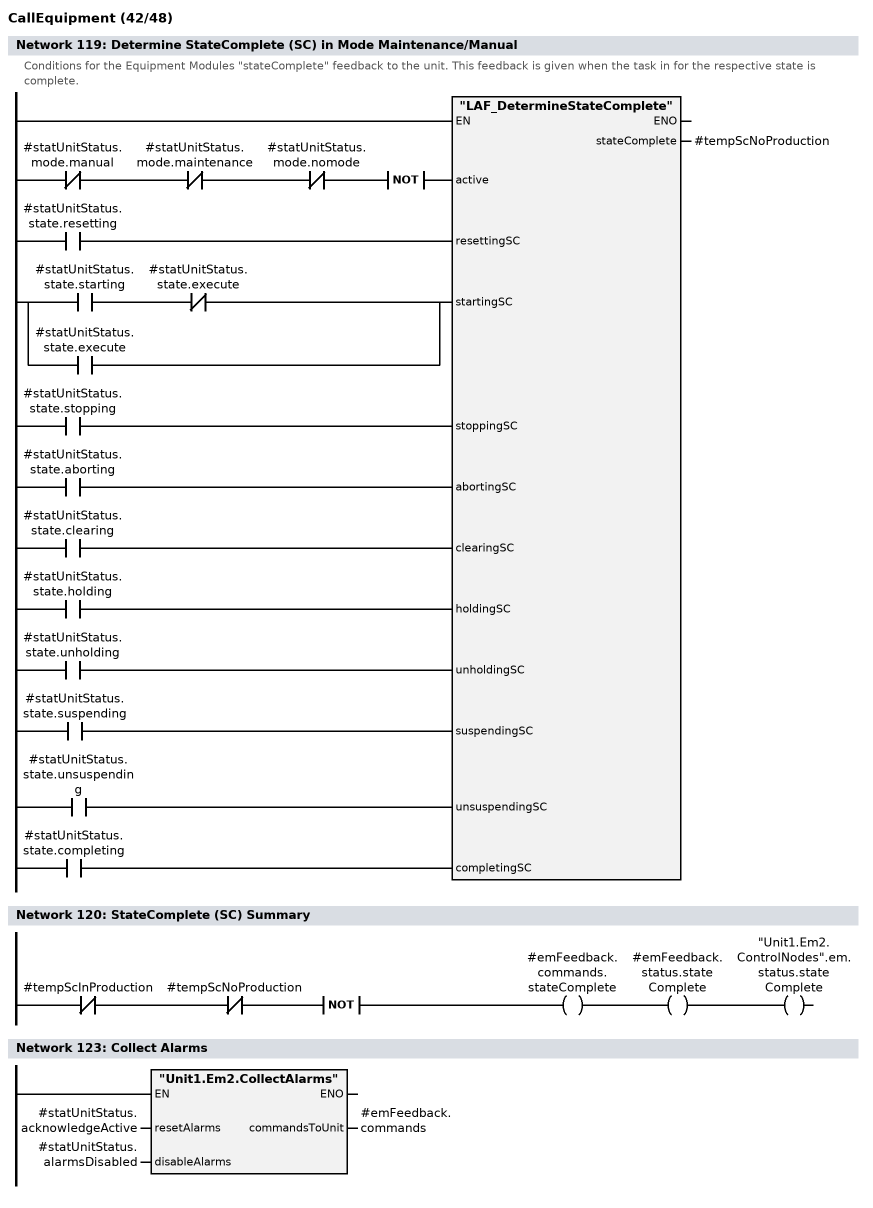
   RUNG wire#powerrail
      "LAF_DetermineStateComplete"(active := wire#w1, resettingSC := wire#w2, startingSC := wire#w3, stoppingSC := wire#w4, abortingSC := wire#w5, clearingSC := wire#w6, holdingSC := wire#w7, unholdingSC := wire#w8, suspendingSC := wire#w9, unsuspendingSC := wire#w10, completingSC := wire#w11, stateComplete => #tempScNoProduction)
   END_RUNG
   RUNG wire#powerrail
      I_Contact( #statUnitStatus.mode.manual )
      I_Contact( #statUnitStatus.mode.maintenance )
      I_Contact( #statUnitStatus.mode.nomode )
      Not()
   END_RUNG wire#w1
   RUNG wire#powerrail
      Contact( #statUnitStatus.state.resetting )
   END_RUNG wire#w2
   RUNG wire#powerrail
      Contact( #statUnitStatus.state.starting )
      I_Contact( #statUnitStatus.state.execute )
   END_RUNG wire#w3
   RUNG wire#powerrail
      Contact( #statUnitStatus.state.execute )
   END_RUNG wire#w3
   RUNG wire#powerrail
      Contact( #statUnitStatus.state.stopping )
   END_RUNG wire#w4
   RUNG wire#powerrail
      Contact( #statUnitStatus.state.aborting )
   END_RUNG wire#w5
   RUNG wire#powerrail
      Contact( #statUnitStatus.state.clearing )
   END_RUNG wire#w6
   RUNG wire#powerrail
      Contact( #statUnitStatus.state.holding )
   END_RUNG wire#w7
   RUNG wire#powerrail
      Contact( #statUnitStatus.state.unholding )
   END_RUNG wire#w8
   RUNG wire#powerrail
      Contact( #statUnitStatus.state.suspending )
   END_RUNG wire#w9
   RUNG wire#powerrail
      Contact( #statUnitStatus.state.unsuspending )
   END_RUNG wire#w10
   RUNG wire#powerrail
      Contact( #statUnitStatus.state.completing )
   END_RUNG wire#w11
   // the same network as SCL:
   "LAF_DetermineStateComplete"(active := NOT (NOT #statUnitStatus.mode.manual AND NOT #statUnitStatus.mode.maintenance AND NOT #statUnitStatus.mode.nomode),
                           resettingSC := #statUnitStatus.state.resetting,
                           startingSC := (#statUnitStatus.state.starting AND NOT #statUnitStatus.state.execute) OR #statUnitStatus.state.execute,
                           stoppingSC := #statUnitStatus.state.stopping,
                           abortingSC := #statUnitStatus.state.aborting,
                           clearingSC := #statUnitStatus.state.clearing,
                           holdingSC := #statUnitStatus.state.holding,
                           unholdingSC := #statUnitStatus.state.unholding,
                           suspendingSC := #statUnitStatus.state.suspending,
                           unsuspendingSC := #statUnitStatus.state.unsuspending,
                           completingSC := #statUnitStatus.state.completing,
                           stateComplete => #tempScNoProduction);
END_REGION

REGION Network 120: StateComplete (SC) Summary
   RUNG wire#powerrail
      I_Contact( #tempScInProduction )
      I_Contact( #tempScNoProduction )
      Not()
      Coil( #emFeedback.commands.stateComplete )
      Coil( #emFeedback.status.stateComplete )
      Coil( "Unit1.Em2.ControlNodes".em.status.stateComplete )
   END_RUNG
   // the same network as SCL:
   #emFeedback.commands.stateComplete := NOT (NOT #tempScInProduction AND NOT #tempScNoProduction);
   #emFeedback.status.stateComplete := #emFeedback.commands.stateComplete;
   "Unit1.Em2.ControlNodes".em.status.stateComplete := #emFeedback.commands.stateComplete;
END_REGION

REGION Network 122: *************** Alarms **********************************
END_REGION

REGION Network 123: Collect Alarms
   RUNG wire#powerrail
      "Unit1.Em2.CollectAlarms"(resetAlarms := #statUnitStatus.acknowledgeActive, disableAlarms := #statUnitStatus.alarmsDisabled, commandsToUnit => #emFeedback.commands)
   END_RUNG
   // the same network as SCL:
   "Unit1.Em2.CollectAlarms"(resetAlarms := #statUnitStatus.acknowledgeActive,
                           disableAlarms := #statUnitStatus.alarmsDisabled,
                           commandsToUnit => #emFeedback.commands);
END_REGION

REGION Network 124: Manage Alarms
   // Derive commands from the ProDiag supervision. The ProDiag supervisions contain categories which define the reaction of these supervisions (e.g. abort, stop, hold). These are handed over as commands to the unit level.
   // Alternatively, if no ProDiag should be used, you can use the LAF_ManageBitAlarms to realize bit alarm handling. This block can be found in LAF in folder 70_AlarmHandling.
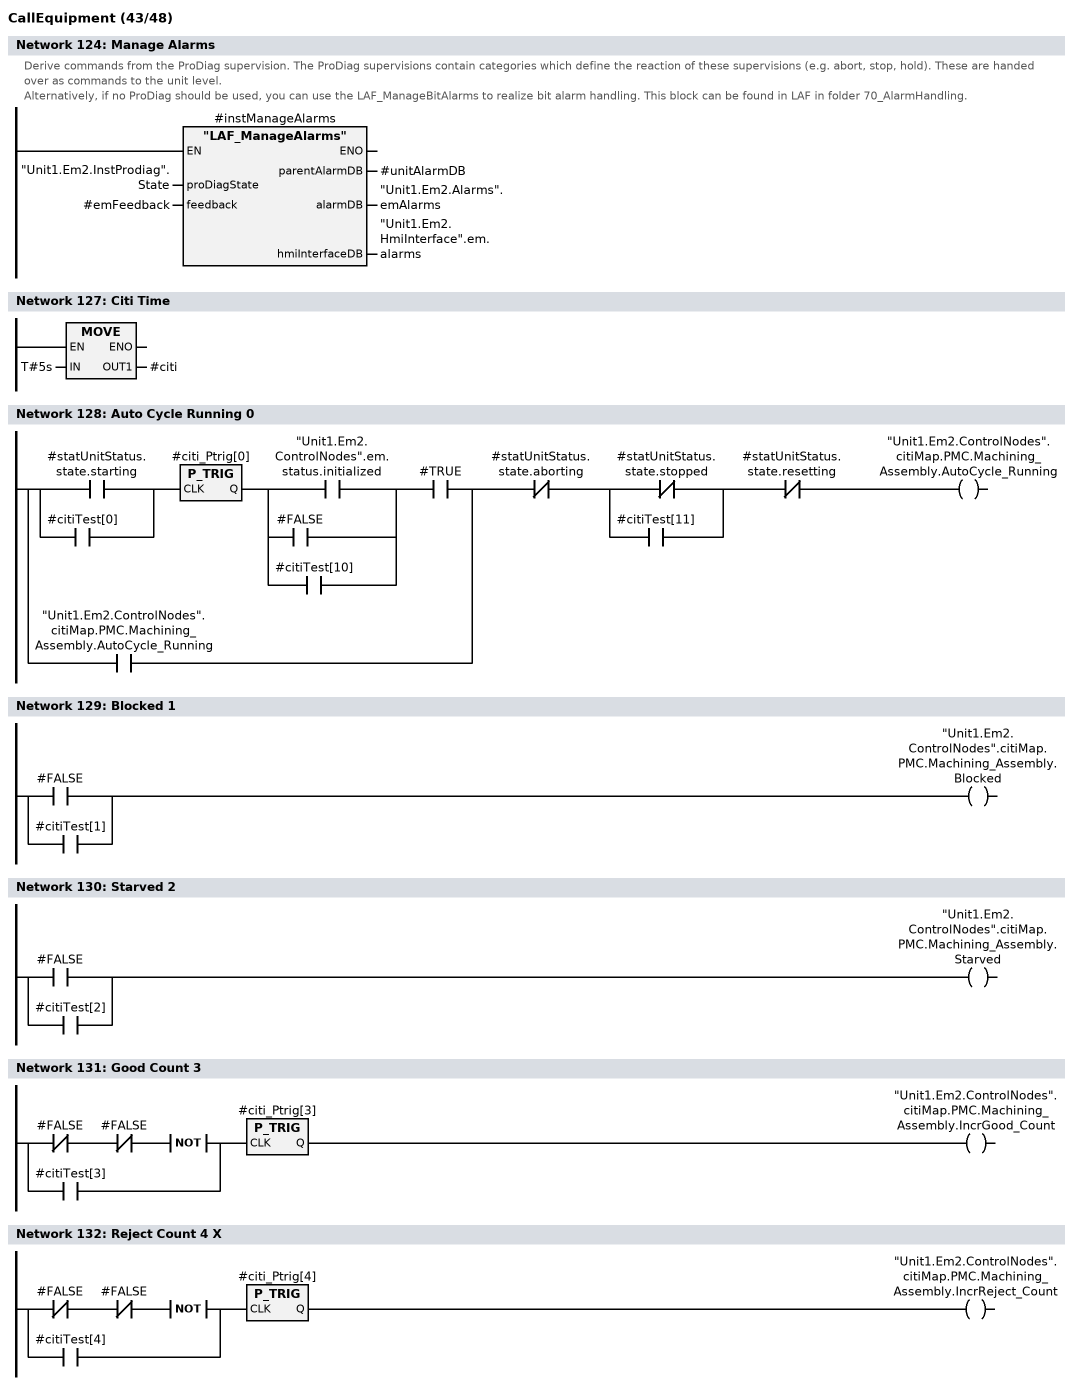
   RUNG wire#powerrail
      #instManageAlarms(proDiagState := "Unit1.Em2.InstProdiag".State, feedback := #emFeedback, parentAlarmDB => #unitAlarmDB, alarmDB => "Unit1.Em2.Alarms".emAlarms, hmiInterfaceDB => "Unit1.Em2.HmiInterface".em.alarms)
   END_RUNG
   // the same network as SCL:
   #instManageAlarms(proDiagState := "Unit1.Em2.InstProdiag".State,   // "LAF_ManageAlarms"
                     feedback := #emFeedback,
                     parentAlarmDB => #unitAlarmDB,
                     alarmDB => "Unit1.Em2.Alarms".emAlarms,
                     hmiInterfaceDB => "Unit1.Em2.HmiInterface".em.alarms);
END_REGION

REGION Network 126: ******************** CITI ********************
END_REGION

REGION Network 127: Citi Time
   RUNG wire#powerrail
      Move(in := T#5s, out1 => #citi)
   END_RUNG
   // the same network as SCL:
   #citi := T#5s;
END_REGION

REGION Network 128: Auto Cycle Running 0
   RUNG wire#powerrail
      Contact( #statUnitStatus.state.starting )
      wire#w1
      P_Trig( #citi_Ptrig[0] )
      wire#w2
      Contact( "Unit1.Em2.ControlNodes".em.status.initialized )
      wire#w3
      Contact( #TRUE )
      wire#w4
      I_Contact( #statUnitStatus.state.aborting )
      wire#w5
      I_Contact( #statUnitStatus.state.stopped )
      wire#w6
      I_Contact( #statUnitStatus.state.resetting )
      Coil( "Unit1.Em2.ControlNodes".citiMap.PMC.Machining_Assembly.AutoCycle_Running )
   END_RUNG
   RUNG wire#powerrail
      Contact( #citiTest[0] )
   END_RUNG wire#w1
   RUNG wire#w2
      Contact( #FALSE )
   END_RUNG wire#w3
   RUNG wire#w2
      Contact( #citiTest[10] )
   END_RUNG wire#w3
   RUNG wire#powerrail
      Contact( "Unit1.Em2.ControlNodes".citiMap.PMC.Machining_Assembly.AutoCycle_Running )
   END_RUNG wire#w4
   RUNG wire#w5
      Contact( #citiTest[11] )
   END_RUNG wire#w6
   // the same network as SCL:
   #_w1 := #statUnitStatus.state.starting OR #citiTest[0];
   #_w2 := #_w1 AND NOT #citi_Ptrig[0];   // rising edge
   #citi_Ptrig[0] := #_w1;
   "Unit1.Em2.ControlNodes".citiMap.PMC.Machining_Assembly.AutoCycle_Running := ((#_w2 AND ("Unit1.Em2.ControlNodes".em.status.initialized OR #FALSE OR #citiTest[10]) AND #TRUE) OR "Unit1.Em2.ControlNodes".citiMap.PMC.Machining_Assembly.AutoCycle_Running) AND NOT #statUnitStatus.state.aborting AND (NOT #statUnitStatus.state.stopped OR #citiTest[11]) AND NOT #statUnitStatus.state.resetting;
END_REGION

REGION Network 129: Blocked 1
   RUNG wire#powerrail
      Contact( #FALSE )
      wire#w1
      Coil( "Unit1.Em2.ControlNodes".citiMap.PMC.Machining_Assembly.Blocked )
   END_RUNG
   RUNG wire#powerrail
      Contact( #citiTest[1] )
   END_RUNG wire#w1
   // the same network as SCL:
   "Unit1.Em2.ControlNodes".citiMap.PMC.Machining_Assembly.Blocked := #FALSE OR #citiTest[1];
END_REGION

REGION Network 130: Starved 2
   RUNG wire#powerrail
      Contact( #FALSE )
      wire#w1
      Coil( "Unit1.Em2.ControlNodes".citiMap.PMC.Machining_Assembly.Starved )
   END_RUNG
   RUNG wire#powerrail
      Contact( #citiTest[2] )
   END_RUNG wire#w1
   // the same network as SCL:
   "Unit1.Em2.ControlNodes".citiMap.PMC.Machining_Assembly.Starved := #FALSE OR #citiTest[2];
END_REGION

REGION Network 131: Good Count 3
   RUNG wire#powerrail
      I_Contact( #FALSE )
      I_Contact( #FALSE )
      Not()
      wire#w1
      P_Trig( #citi_Ptrig[3] )
      Coil( "Unit1.Em2.ControlNodes".citiMap.PMC.Machining_Assembly.IncrGood_Count )
   END_RUNG
   RUNG wire#powerrail
      Contact( #citiTest[3] )
   END_RUNG wire#w1
   // the same network as SCL:
   #_w1 := NOT (NOT #FALSE AND NOT #FALSE) OR #citiTest[3];
   #_w2 := #_w1 AND NOT #citi_Ptrig[3];   // rising edge
   #citi_Ptrig[3] := #_w1;
   "Unit1.Em2.ControlNodes".citiMap.PMC.Machining_Assembly.IncrGood_Count := #_w2;
END_REGION

REGION Network 132: Reject Count 4 X
   RUNG wire#powerrail
      I_Contact( #FALSE )
      I_Contact( #FALSE )
      Not()
      wire#w1
      P_Trig( #citi_Ptrig[4] )
      Coil( "Unit1.Em2.ControlNodes".citiMap.PMC.Machining_Assembly.IncrReject_Count )
   END_RUNG
   RUNG wire#powerrail
      Contact( #citiTest[4] )
   END_RUNG wire#w1
   // the same network as SCL:
   #_w1 := NOT (NOT #FALSE AND NOT #FALSE) OR #citiTest[4];
   #_w2 := #_w1 AND NOT #citi_Ptrig[4];   // rising edge
   #citi_Ptrig[4] := #_w1;
   "Unit1.Em2.ControlNodes".citiMap.PMC.Machining_Assembly.IncrReject_Count := #_w2;
END_REGION

REGION Network 133: Cycle End Trigger 5
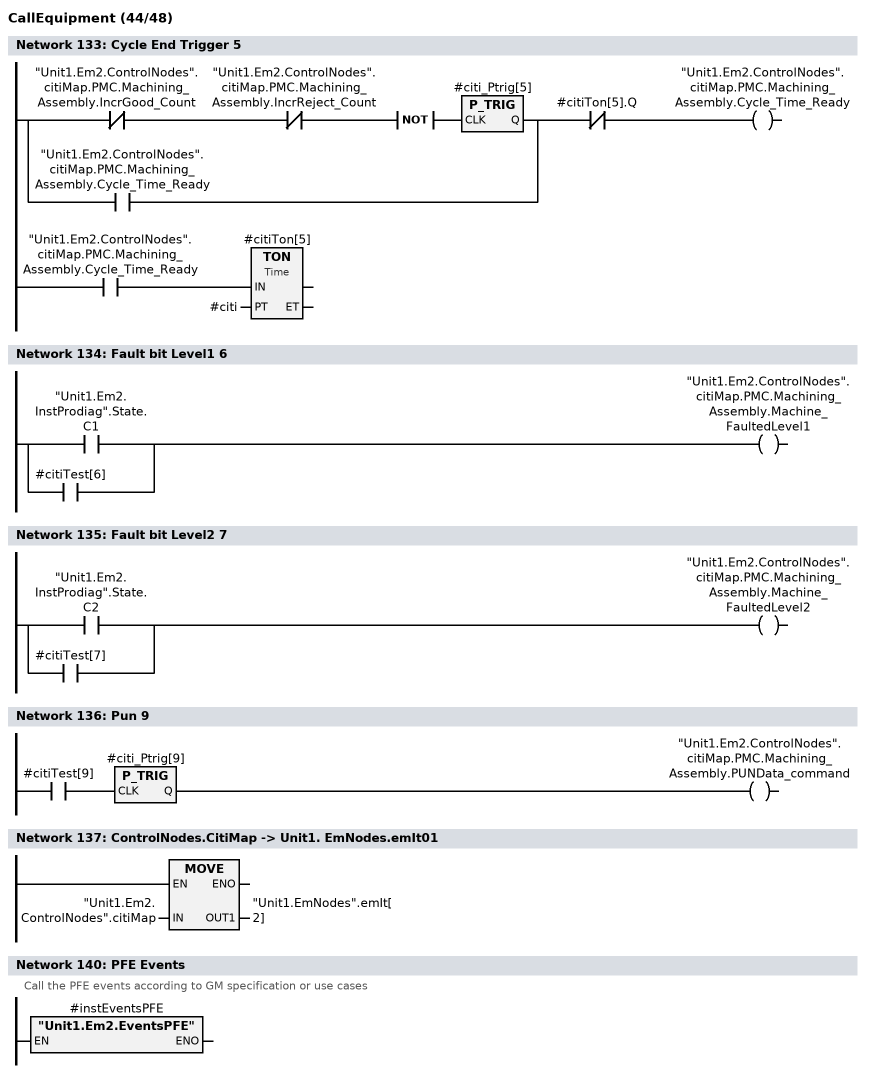
   RUNG wire#powerrail
      I_Contact( "Unit1.Em2.ControlNodes".citiMap.PMC.Machining_Assembly.IncrGood_Count )
      I_Contact( "Unit1.Em2.ControlNodes".citiMap.PMC.Machining_Assembly.IncrReject_Count )
      Not()
      P_Trig( #citi_Ptrig[5] )
      wire#w1
      I_Contact( #citiTon[5].Q )
      Coil( "Unit1.Em2.ControlNodes".citiMap.PMC.Machining_Assembly.Cycle_Time_Ready )
   END_RUNG
   RUNG wire#powerrail
      Contact( "Unit1.Em2.ControlNodes".citiMap.PMC.Machining_Assembly.Cycle_Time_Ready )
   END_RUNG wire#w1
   RUNG wire#powerrail
      Contact( "Unit1.Em2.ControlNodes".citiMap.PMC.Machining_Assembly.Cycle_Time_Ready )
      { S7_Templates := "time_type := Time" } #citiTon[5].TON(pt := #citi, et =>)
   END_RUNG
   // the same network as SCL:
   #_w1 := NOT (NOT "Unit1.Em2.ControlNodes".citiMap.PMC.Machining_Assembly.IncrGood_Count AND NOT "Unit1.Em2.ControlNodes".citiMap.PMC.Machining_Assembly.IncrReject_Count);
   #_w2 := #_w1 AND NOT #citi_Ptrig[5];   // rising edge
   #citi_Ptrig[5] := #_w1;
   "Unit1.Em2.ControlNodes".citiMap.PMC.Machining_Assembly.Cycle_Time_Ready := (#_w2 OR "Unit1.Em2.ControlNodes".citiMap.PMC.Machining_Assembly.Cycle_Time_Ready) AND NOT #citiTon[5].Q;
   #citiTon[5].TON(IN := "Unit1.Em2.ControlNodes".citiMap.PMC.Machining_Assembly.Cycle_Time_Ready, PT := #citi);
END_REGION

REGION Network 134: Fault bit Level1 6
   RUNG wire#powerrail
      Contact( "Unit1.Em2.InstProdiag".State.C1 )
      wire#w1
      Coil( "Unit1.Em2.ControlNodes".citiMap.PMC.Machining_Assembly.Machine_FaultedLevel1 )
   END_RUNG
   RUNG wire#powerrail
      Contact( #citiTest[6] )
   END_RUNG wire#w1
   // the same network as SCL:
   "Unit1.Em2.ControlNodes".citiMap.PMC.Machining_Assembly.Machine_FaultedLevel1 := "Unit1.Em2.InstProdiag".State.C1 OR #citiTest[6];
END_REGION

REGION Network 135: Fault bit Level2 7
   RUNG wire#powerrail
      Contact( "Unit1.Em2.InstProdiag".State.C2 )
      wire#w1
      Coil( "Unit1.Em2.ControlNodes".citiMap.PMC.Machining_Assembly.Machine_FaultedLevel2 )
   END_RUNG
   RUNG wire#powerrail
      Contact( #citiTest[7] )
   END_RUNG wire#w1
   // the same network as SCL:
   "Unit1.Em2.ControlNodes".citiMap.PMC.Machining_Assembly.Machine_FaultedLevel2 := "Unit1.Em2.InstProdiag".State.C2 OR #citiTest[7];
END_REGION

REGION Network 136: Pun 9
   RUNG wire#powerrail
      Contact( #citiTest[9] )
      P_Trig( #citi_Ptrig[9] )
      Coil( "Unit1.Em2.ControlNodes".citiMap.PMC.Machining_Assembly.PUNData_command )
   END_RUNG
   // the same network as SCL:
   #_w1 := #citiTest[9] AND NOT #citi_Ptrig[9];   // rising edge
   #citi_Ptrig[9] := #citiTest[9];
   "Unit1.Em2.ControlNodes".citiMap.PMC.Machining_Assembly.PUNData_command := #_w1;
END_REGION

REGION Network 137: ControlNodes.CitiMap -> Unit1. EmNodes.emIt01
   RUNG wire#powerrail
      Move(in := "Unit1.Em2.ControlNodes".citiMap, out1 => "Unit1.EmNodes".emIt[2])
   END_RUNG
   // the same network as SCL:
   "Unit1.EmNodes".emIt[2] := "Unit1.Em2.ControlNodes".citiMap;
END_REGION

REGION Network 139: *************** PFE Events**********************************
END_REGION

REGION Network 140: PFE Events
   // Call the PFE events according to GM specification or use cases
   RUNG wire#powerrail
      #instEventsPFE()
   END_RUNG
   // the same network as SCL:
   #instEventsPFE();   // "Unit1.Em2.EventsPFE"
END_REGION

REGION Network 142: ******************** Unit Output ********************
END_REGION

REGION Network 143: Em2 Relations Softcam
END_REGION

REGION Network 144: Em2 Relations Home Check
END_REGION

REGION Network 145: Em2 Relations Cm Status Cylinder
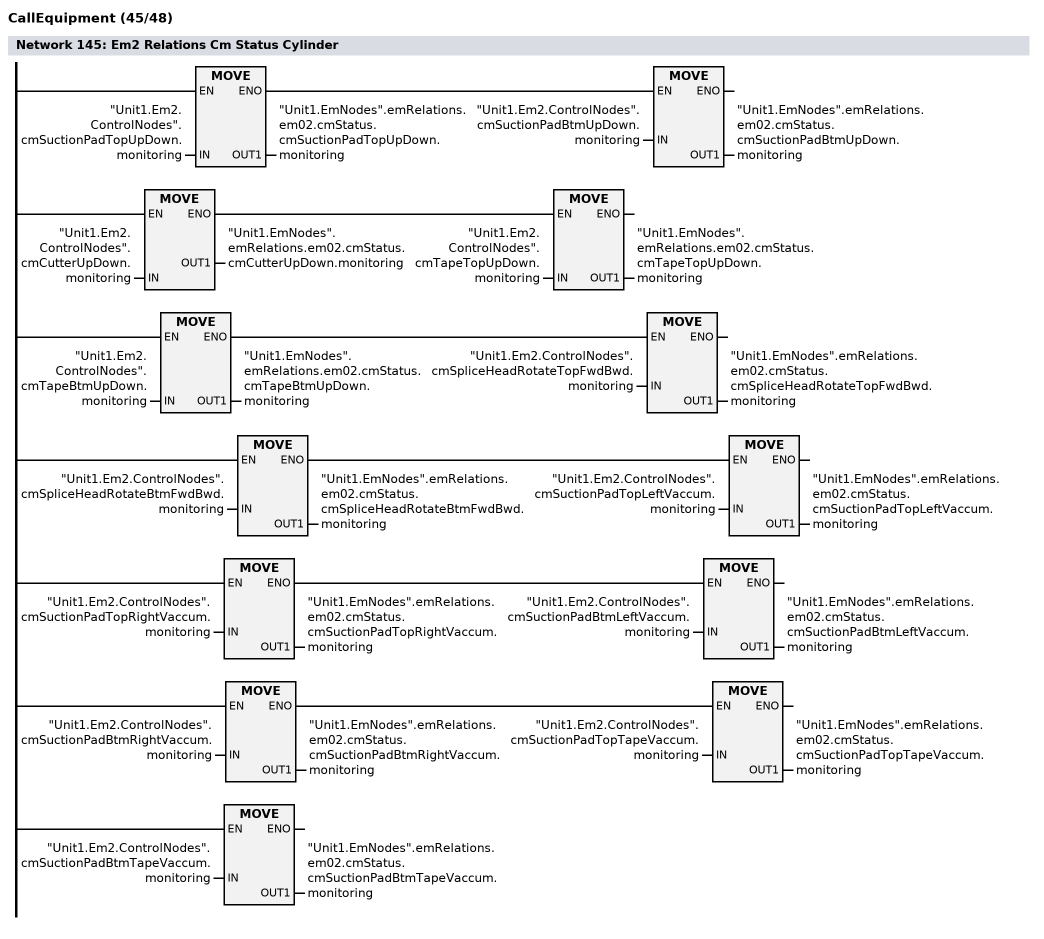
   RUNG wire#powerrail
      Move(in := "Unit1.Em2.ControlNodes".cmSuctionPadTopUpDown.monitoring, out1 => "Unit1.EmNodes".emRelations.em02.cmStatus.cmSuctionPadTopUpDown.monitoring)
      Move(in := "Unit1.Em2.ControlNodes".cmSuctionPadBtmUpDown.monitoring, out1 => "Unit1.EmNodes".emRelations.em02.cmStatus.cmSuctionPadBtmUpDown.monitoring)
   END_RUNG
   RUNG wire#powerrail
      Move(in := "Unit1.Em2.ControlNodes".cmCutterUpDown.monitoring, out1 => "Unit1.EmNodes".emRelations.em02.cmStatus.cmCutterUpDown.monitoring)
      Move(in := "Unit1.Em2.ControlNodes".cmTapeTopUpDown.monitoring, out1 => "Unit1.EmNodes".emRelations.em02.cmStatus.cmTapeTopUpDown.monitoring)
   END_RUNG
   RUNG wire#powerrail
      Move(in := "Unit1.Em2.ControlNodes".cmTapeBtmUpDown.monitoring, out1 => "Unit1.EmNodes".emRelations.em02.cmStatus.cmTapeBtmUpDown.monitoring)
      Move(in := "Unit1.Em2.ControlNodes".cmSpliceHeadRotateTopFwdBwd.monitoring, out1 => "Unit1.EmNodes".emRelations.em02.cmStatus.cmSpliceHeadRotateTopFwdBwd.monitoring)
   END_RUNG
   RUNG wire#powerrail
      Move(in := "Unit1.Em2.ControlNodes".cmSpliceHeadRotateBtmFwdBwd.monitoring, out1 => "Unit1.EmNodes".emRelations.em02.cmStatus.cmSpliceHeadRotateBtmFwdBwd.monitoring)
      Move(in := "Unit1.Em2.ControlNodes".cmSuctionPadTopLeftVaccum.monitoring, out1 => "Unit1.EmNodes".emRelations.em02.cmStatus.cmSuctionPadTopLeftVaccum.monitoring)
   END_RUNG
   RUNG wire#powerrail
      Move(in := "Unit1.Em2.ControlNodes".cmSuctionPadTopRightVaccum.monitoring, out1 => "Unit1.EmNodes".emRelations.em02.cmStatus.cmSuctionPadTopRightVaccum.monitoring)
      Move(in := "Unit1.Em2.ControlNodes".cmSuctionPadBtmLeftVaccum.monitoring, out1 => "Unit1.EmNodes".emRelations.em02.cmStatus.cmSuctionPadBtmLeftVaccum.monitoring)
   END_RUNG
   RUNG wire#powerrail
      Move(in := "Unit1.Em2.ControlNodes".cmSuctionPadBtmRightVaccum.monitoring, out1 => "Unit1.EmNodes".emRelations.em02.cmStatus.cmSuctionPadBtmRightVaccum.monitoring)
      Move(in := "Unit1.Em2.ControlNodes".cmSuctionPadTopTapeVaccum.monitoring, out1 => "Unit1.EmNodes".emRelations.em02.cmStatus.cmSuctionPadTopTapeVaccum.monitoring)
   END_RUNG
   RUNG wire#powerrail
      Move(in := "Unit1.Em2.ControlNodes".cmSuctionPadBtmTapeVaccum.monitoring, out1 => "Unit1.EmNodes".emRelations.em02.cmStatus.cmSuctionPadBtmTapeVaccum.monitoring)
   END_RUNG
   // the same network as SCL:
   "Unit1.EmNodes".emRelations.em02.cmStatus.cmSuctionPadTopUpDown.monitoring := "Unit1.Em2.ControlNodes".cmSuctionPadTopUpDown.monitoring;
   "Unit1.EmNodes".emRelations.em02.cmStatus.cmSuctionPadBtmUpDown.monitoring := "Unit1.Em2.ControlNodes".cmSuctionPadBtmUpDown.monitoring;
   "Unit1.EmNodes".emRelations.em02.cmStatus.cmCutterUpDown.monitoring := "Unit1.Em2.ControlNodes".cmCutterUpDown.monitoring;
   "Unit1.EmNodes".emRelations.em02.cmStatus.cmTapeTopUpDown.monitoring := "Unit1.Em2.ControlNodes".cmTapeTopUpDown.monitoring;
   "Unit1.EmNodes".emRelations.em02.cmStatus.cmTapeBtmUpDown.monitoring := "Unit1.Em2.ControlNodes".cmTapeBtmUpDown.monitoring;
   "Unit1.EmNodes".emRelations.em02.cmStatus.cmSpliceHeadRotateTopFwdBwd.monitoring := "Unit1.Em2.ControlNodes".cmSpliceHeadRotateTopFwdBwd.monitoring;
   "Unit1.EmNodes".emRelations.em02.cmStatus.cmSpliceHeadRotateBtmFwdBwd.monitoring := "Unit1.Em2.ControlNodes".cmSpliceHeadRotateBtmFwdBwd.monitoring;
   "Unit1.EmNodes".emRelations.em02.cmStatus.cmSuctionPadTopLeftVaccum.monitoring := "Unit1.Em2.ControlNodes".cmSuctionPadTopLeftVaccum.monitoring;
   "Unit1.EmNodes".emRelations.em02.cmStatus.cmSuctionPadTopRightVaccum.monitoring := "Unit1.Em2.ControlNodes".cmSuctionPadTopRightVaccum.monitoring;
   "Unit1.EmNodes".emRelations.em02.cmStatus.cmSuctionPadBtmLeftVaccum.monitoring := "Unit1.Em2.ControlNodes".cmSuctionPadBtmLeftVaccum.monitoring;
   "Unit1.EmNodes".emRelations.em02.cmStatus.cmSuctionPadBtmRightVaccum.monitoring := "Unit1.Em2.ControlNodes".cmSuctionPadBtmRightVaccum.monitoring;
   "Unit1.EmNodes".emRelations.em02.cmStatus.cmSuctionPadTopTapeVaccum.monitoring := "Unit1.Em2.ControlNodes".cmSuctionPadTopTapeVaccum.monitoring;
   "Unit1.EmNodes".emRelations.em02.cmStatus.cmSuctionPadBtmTapeVaccum.monitoring := "Unit1.Em2.ControlNodes".cmSuctionPadBtmTapeVaccum.monitoring;
END_REGION

REGION Network 146: Em2 Relations CmStatus Digital Signal
END_REGION

REGION Network 147: Em2 Relations Select Job Status
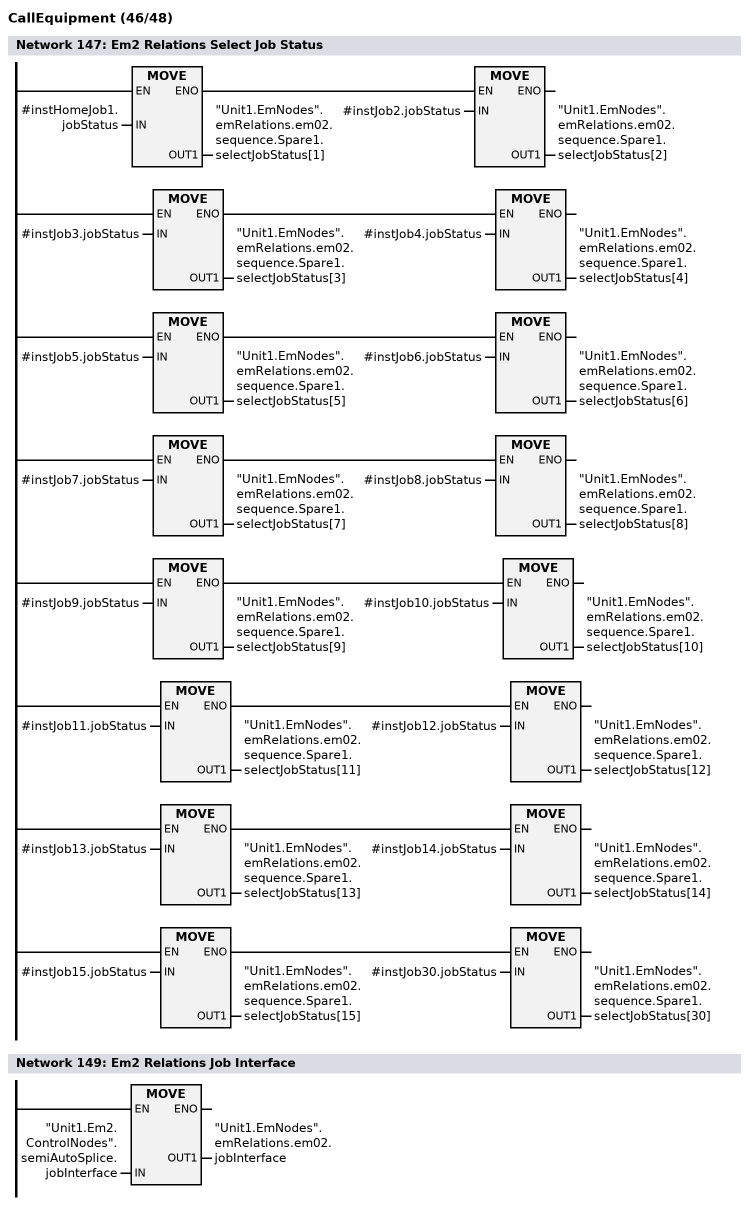
   RUNG wire#powerrail
      Move(in := #instHomeJob1.jobStatus, out1 => "Unit1.EmNodes".emRelations.em02.sequence.Spare1.selectJobStatus[1])
      Move(in := #instJob2.jobStatus, out1 => "Unit1.EmNodes".emRelations.em02.sequence.Spare1.selectJobStatus[2])
   END_RUNG
   RUNG wire#powerrail
      Move(in := #instJob3.jobStatus, out1 => "Unit1.EmNodes".emRelations.em02.sequence.Spare1.selectJobStatus[3])
      Move(in := #instJob4.jobStatus, out1 => "Unit1.EmNodes".emRelations.em02.sequence.Spare1.selectJobStatus[4])
   END_RUNG
   RUNG wire#powerrail
      Move(in := #instJob5.jobStatus, out1 => "Unit1.EmNodes".emRelations.em02.sequence.Spare1.selectJobStatus[5])
      Move(in := #instJob6.jobStatus, out1 => "Unit1.EmNodes".emRelations.em02.sequence.Spare1.selectJobStatus[6])
   END_RUNG
   RUNG wire#powerrail
      Move(in := #instJob7.jobStatus, out1 => "Unit1.EmNodes".emRelations.em02.sequence.Spare1.selectJobStatus[7])
      Move(in := #instJob8.jobStatus, out1 => "Unit1.EmNodes".emRelations.em02.sequence.Spare1.selectJobStatus[8])
   END_RUNG
   RUNG wire#powerrail
      Move(in := #instJob9.jobStatus, out1 => "Unit1.EmNodes".emRelations.em02.sequence.Spare1.selectJobStatus[9])
      Move(in := #instJob10.jobStatus, out1 => "Unit1.EmNodes".emRelations.em02.sequence.Spare1.selectJobStatus[10])
   END_RUNG
   RUNG wire#powerrail
      Move(in := #instJob11.jobStatus, out1 => "Unit1.EmNodes".emRelations.em02.sequence.Spare1.selectJobStatus[11])
      Move(in := #instJob12.jobStatus, out1 => "Unit1.EmNodes".emRelations.em02.sequence.Spare1.selectJobStatus[12])
   END_RUNG
   RUNG wire#powerrail
      Move(in := #instJob13.jobStatus, out1 => "Unit1.EmNodes".emRelations.em02.sequence.Spare1.selectJobStatus[13])
      Move(in := #instJob14.jobStatus, out1 => "Unit1.EmNodes".emRelations.em02.sequence.Spare1.selectJobStatus[14])
   END_RUNG
   RUNG wire#powerrail
      Move(in := #instJob15.jobStatus, out1 => "Unit1.EmNodes".emRelations.em02.sequence.Spare1.selectJobStatus[15])
      Move(in := #instJob30.jobStatus, out1 => "Unit1.EmNodes".emRelations.em02.sequence.Spare1.selectJobStatus[30])
   END_RUNG
   // the same network as SCL:
   "Unit1.EmNodes".emRelations.em02.sequence.Spare1.selectJobStatus[1] := #instHomeJob1.jobStatus;
   "Unit1.EmNodes".emRelations.em02.sequence.Spare1.selectJobStatus[2] := #instJob2.jobStatus;
   "Unit1.EmNodes".emRelations.em02.sequence.Spare1.selectJobStatus[3] := #instJob3.jobStatus;
   "Unit1.EmNodes".emRelations.em02.sequence.Spare1.selectJobStatus[4] := #instJob4.jobStatus;
   "Unit1.EmNodes".emRelations.em02.sequence.Spare1.selectJobStatus[5] := #instJob5.jobStatus;
   "Unit1.EmNodes".emRelations.em02.sequence.Spare1.selectJobStatus[6] := #instJob6.jobStatus;
   "Unit1.EmNodes".emRelations.em02.sequence.Spare1.selectJobStatus[7] := #instJob7.jobStatus;
   "Unit1.EmNodes".emRelations.em02.sequence.Spare1.selectJobStatus[8] := #instJob8.jobStatus;
   "Unit1.EmNodes".emRelations.em02.sequence.Spare1.selectJobStatus[9] := #instJob9.jobStatus;
   "Unit1.EmNodes".emRelations.em02.sequence.Spare1.selectJobStatus[10] := #instJob10.jobStatus;
   "Unit1.EmNodes".emRelations.em02.sequence.Spare1.selectJobStatus[11] := #instJob11.jobStatus;
   "Unit1.EmNodes".emRelations.em02.sequence.Spare1.selectJobStatus[12] := #instJob12.jobStatus;
   "Unit1.EmNodes".emRelations.em02.sequence.Spare1.selectJobStatus[13] := #instJob13.jobStatus;
   "Unit1.EmNodes".emRelations.em02.sequence.Spare1.selectJobStatus[14] := #instJob14.jobStatus;
   "Unit1.EmNodes".emRelations.em02.sequence.Spare1.selectJobStatus[15] := #instJob15.jobStatus;
   "Unit1.EmNodes".emRelations.em02.sequence.Spare1.selectJobStatus[30] := #instJob30.jobStatus;
END_REGION

REGION Network 148: Em2 Relations Sequence Interface
END_REGION

REGION Network 149: Em2 Relations Job Interface
   RUNG wire#powerrail
      Move(in := "Unit1.Em2.ControlNodes".semiAutoSplice.jobInterface, out1 => "Unit1.EmNodes".emRelations.em02.jobInterface)
   END_RUNG
   // the same network as SCL:
   "Unit1.EmNodes".emRelations.em02.jobInterface := "Unit1.Em2.ControlNodes".semiAutoSplice.jobInterface;
END_REGION

REGION Network 151: Cylinder
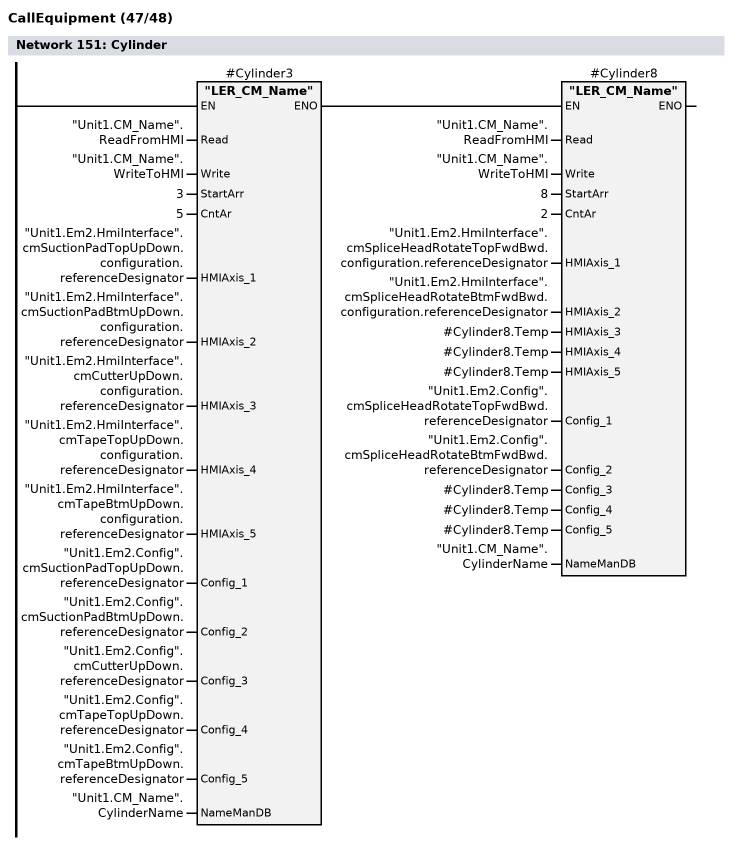
   RUNG wire#powerrail
      #Cylinder3(Read := "Unit1.CM_Name".ReadFromHMI, Write := "Unit1.CM_Name".WriteToHMI, StartArr := 3, CntAr := 5, HMIAxis_1 := "Unit1.Em2.HmiInterface".cmSuctionPadTopUpDown.configuration.referenceDesignator, HMIAxis_2 := "Unit1.Em2.HmiInterface".cmSuctionPadBtmUpDown.configuration.referenceDesignator, HMIAxis_3 := "Unit1.Em2.HmiInterface".cmCutterUpDown.configuration.referenceDesignator, HMIAxis_4 := "Unit1.Em2.HmiInterface".cmTapeTopUpDown.configuration.referenceDesignator, HMIAxis_5 := "Unit1.Em2.HmiInterface".cmTapeBtmUpDown.configuration.referenceDesignator, Config_1 := "Unit1.Em2.Config".cmSuctionPadTopUpDown.referenceDesignator, Config_2 := "Unit1.Em2.Config".cmSuctionPadBtmUpDown.referenceDesignator, Config_3 := "Unit1.Em2.Config".cmCutterUpDown.referenceDesignator, Config_4 := "Unit1.Em2.Config".cmTapeTopUpDown.referenceDesignator, Config_5 := "Unit1.Em2.Config".cmTapeBtmUpDown.referenceDesignator, NameManDB := "Unit1.CM_Name".CylinderName)
      #Cylinder8(Read := "Unit1.CM_Name".ReadFromHMI, Write := "Unit1.CM_Name".WriteToHMI, StartArr := 8, CntAr := 2, HMIAxis_1 := "Unit1.Em2.HmiInterface".cmSpliceHeadRotateTopFwdBwd.configuration.referenceDesignator, HMIAxis_2 := "Unit1.Em2.HmiInterface".cmSpliceHeadRotateBtmFwdBwd.configuration.referenceDesignator, HMIAxis_3 := #Cylinder8.Temp, HMIAxis_4 := #Cylinder8.Temp, HMIAxis_5 := #Cylinder8.Temp, Config_1 := "Unit1.Em2.Config".cmSpliceHeadRotateTopFwdBwd.referenceDesignator, Config_2 := "Unit1.Em2.Config".cmSpliceHeadRotateBtmFwdBwd.referenceDesignator, Config_3 := #Cylinder8.Temp, Config_4 := #Cylinder8.Temp, Config_5 := #Cylinder8.Temp, NameManDB := "Unit1.CM_Name".CylinderName)
   END_RUNG
   // the same network as SCL:
   #Cylinder3(Read := "Unit1.CM_Name".ReadFromHMI,   // "LER_CM_Name"
              Write := "Unit1.CM_Name".WriteToHMI,
              StartArr := 3,
              CntAr := 5,
              HMIAxis_1 := "Unit1.Em2.HmiInterface".cmSuctionPadTopUpDown.configuration.referenceDesignator,
              HMIAxis_2 := "Unit1.Em2.HmiInterface".cmSuctionPadBtmUpDown.configuration.referenceDesignator,
              HMIAxis_3 := "Unit1.Em2.HmiInterface".cmCutterUpDown.configuration.referenceDesignator,
              HMIAxis_4 := "Unit1.Em2.HmiInterface".cmTapeTopUpDown.configuration.referenceDesignator,
              HMIAxis_5 := "Unit1.Em2.HmiInterface".cmTapeBtmUpDown.configuration.referenceDesignator,
              Config_1 := "Unit1.Em2.Config".cmSuctionPadTopUpDown.referenceDesignator,
              Config_2 := "Unit1.Em2.Config".cmSuctionPadBtmUpDown.referenceDesignator,
              Config_3 := "Unit1.Em2.Config".cmCutterUpDown.referenceDesignator,
              Config_4 := "Unit1.Em2.Config".cmTapeTopUpDown.referenceDesignator,
              Config_5 := "Unit1.Em2.Config".cmTapeBtmUpDown.referenceDesignator,
              NameManDB := "Unit1.CM_Name".CylinderName,
              ENO => #_w1);
   IF #_w1 THEN
       #Cylinder8(Read := "Unit1.CM_Name".ReadFromHMI,   // "LER_CM_Name"
                  Write := "Unit1.CM_Name".WriteToHMI,
                  StartArr := 8,
                  CntAr := 2,
                  HMIAxis_1 := "Unit1.Em2.HmiInterface".cmSpliceHeadRotateTopFwdBwd.configuration.referenceDesignator,
                  HMIAxis_2 := "Unit1.Em2.HmiInterface".cmSpliceHeadRotateBtmFwdBwd.configuration.referenceDesignator,
                  HMIAxis_3 := #Cylinder8.Temp,
                  HMIAxis_4 := #Cylinder8.Temp,
                  HMIAxis_5 := #Cylinder8.Temp,
                  Config_1 := "Unit1.Em2.Config".cmSpliceHeadRotateTopFwdBwd.referenceDesignator,
                  Config_2 := "Unit1.Em2.Config".cmSpliceHeadRotateBtmFwdBwd.referenceDesignator,
                  Config_3 := #Cylinder8.Temp,
                  Config_4 := #Cylinder8.Temp,
                  Config_5 := #Cylinder8.Temp,
                  NameManDB := "Unit1.CM_Name".CylinderName);
   END_IF;
END_REGION

REGION Network 152: Cylinder
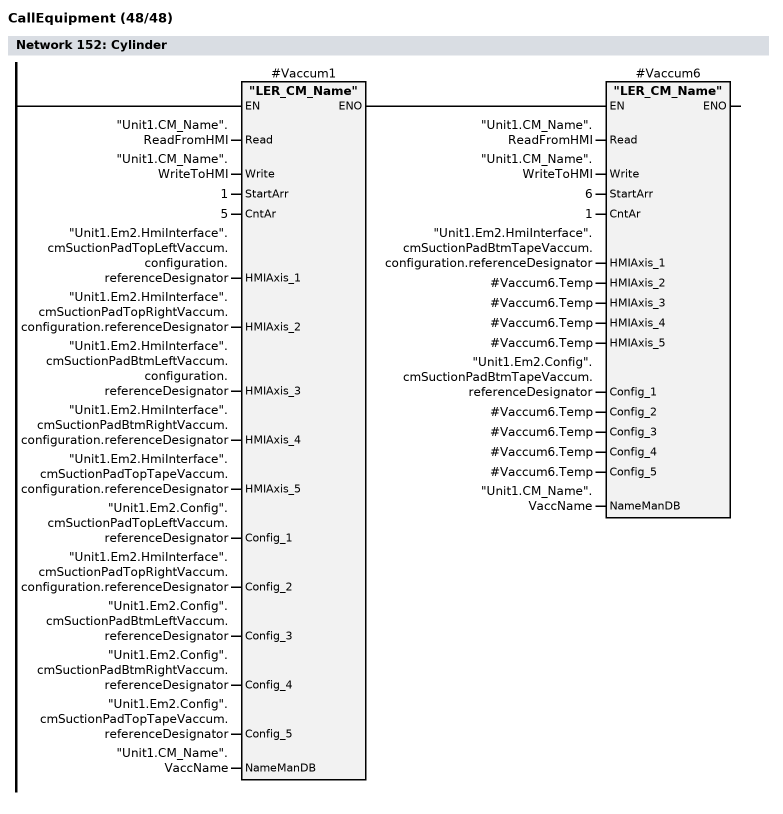
   RUNG wire#powerrail
      #Vaccum1(Read := "Unit1.CM_Name".ReadFromHMI, Write := "Unit1.CM_Name".WriteToHMI, StartArr := 1, CntAr := 5, HMIAxis_1 := "Unit1.Em2.HmiInterface".cmSuctionPadTopLeftVaccum.configuration.referenceDesignator, HMIAxis_2 := "Unit1.Em2.HmiInterface".cmSuctionPadTopRightVaccum.configuration.referenceDesignator, HMIAxis_3 := "Unit1.Em2.HmiInterface".cmSuctionPadBtmLeftVaccum.configuration.referenceDesignator, HMIAxis_4 := "Unit1.Em2.HmiInterface".cmSuctionPadBtmRightVaccum.configuration.referenceDesignator, HMIAxis_5 := "Unit1.Em2.HmiInterface".cmSuctionPadTopTapeVaccum.configuration.referenceDesignator, Config_1 := "Unit1.Em2.Config".cmSuctionPadTopLeftVaccum.referenceDesignator, Config_2 := "Unit1.Em2.HmiInterface".cmSuctionPadTopRightVaccum.configuration.referenceDesignator, Config_3 := "Unit1.Em2.Config".cmSuctionPadBtmLeftVaccum.referenceDesignator, Config_4 := "Unit1.Em2.Config".cmSuctionPadBtmRightVaccum.referenceDesignator, Config_5 := "Unit1.Em2.Config".cmSuctionPadTopTapeVaccum.referenceDesignator, NameManDB := "Unit1.CM_Name".VaccName)
      #Vaccum6(Read := "Unit1.CM_Name".ReadFromHMI, Write := "Unit1.CM_Name".WriteToHMI, StartArr := 6, CntAr := 1, HMIAxis_1 := "Unit1.Em2.HmiInterface".cmSuctionPadBtmTapeVaccum.configuration.referenceDesignator, HMIAxis_2 := #Vaccum6.Temp, HMIAxis_3 := #Vaccum6.Temp, HMIAxis_4 := #Vaccum6.Temp, HMIAxis_5 := #Vaccum6.Temp, Config_1 := "Unit1.Em2.Config".cmSuctionPadBtmTapeVaccum.referenceDesignator, Config_2 := #Vaccum6.Temp, Config_3 := #Vaccum6.Temp, Config_4 := #Vaccum6.Temp, Config_5 := #Vaccum6.Temp, NameManDB := "Unit1.CM_Name".VaccName)
   END_RUNG
   // the same network as SCL:
   #Vaccum1(Read := "Unit1.CM_Name".ReadFromHMI,   // "LER_CM_Name"
            Write := "Unit1.CM_Name".WriteToHMI,
            StartArr := 1,
            CntAr := 5,
            HMIAxis_1 := "Unit1.Em2.HmiInterface".cmSuctionPadTopLeftVaccum.configuration.referenceDesignator,
            HMIAxis_2 := "Unit1.Em2.HmiInterface".cmSuctionPadTopRightVaccum.configuration.referenceDesignator,
            HMIAxis_3 := "Unit1.Em2.HmiInterface".cmSuctionPadBtmLeftVaccum.configuration.referenceDesignator,
            HMIAxis_4 := "Unit1.Em2.HmiInterface".cmSuctionPadBtmRightVaccum.configuration.referenceDesignator,
            HMIAxis_5 := "Unit1.Em2.HmiInterface".cmSuctionPadTopTapeVaccum.configuration.referenceDesignator,
            Config_1 := "Unit1.Em2.Config".cmSuctionPadTopLeftVaccum.referenceDesignator,
            Config_2 := "Unit1.Em2.HmiInterface".cmSuctionPadTopRightVaccum.configuration.referenceDesignator,
            Config_3 := "Unit1.Em2.Config".cmSuctionPadBtmLeftVaccum.referenceDesignator,
            Config_4 := "Unit1.Em2.Config".cmSuctionPadBtmRightVaccum.referenceDesignator,
            Config_5 := "Unit1.Em2.Config".cmSuctionPadTopTapeVaccum.referenceDesignator,
            NameManDB := "Unit1.CM_Name".VaccName,
            ENO => #_w1);
   IF #_w1 THEN
       #Vaccum6(Read := "Unit1.CM_Name".ReadFromHMI,   // "LER_CM_Name"
                Write := "Unit1.CM_Name".WriteToHMI,
                StartArr := 6,
                CntAr := 1,
                HMIAxis_1 := "Unit1.Em2.HmiInterface".cmSuctionPadBtmTapeVaccum.configuration.referenceDesignator,
                HMIAxis_2 := #Vaccum6.Temp,
                HMIAxis_3 := #Vaccum6.Temp,
                HMIAxis_4 := #Vaccum6.Temp,
                HMIAxis_5 := #Vaccum6.Temp,
                Config_1 := "Unit1.Em2.Config".cmSuctionPadBtmTapeVaccum.referenceDesignator,
                Config_2 := #Vaccum6.Temp,
                Config_3 := #Vaccum6.Temp,
                Config_4 := #Vaccum6.Temp,
                Config_5 := #Vaccum6.Temp,
                NameManDB := "Unit1.CM_Name".VaccName);
   END_IF;
END_REGION

REGION Network 153: -----------------------------------------------------------------
END_REGION
END_FUNCTION_BLOCK
